{attribute 'GeneratedUsingTerminal: EL7411-0000-0016'}
{attribute addProperty BoxType "EL7411-0000-0016"}
{attribute addProperty Id "AdsAddrAT %I*AMSADDR8DcOutputShiftAT %I*DINT4DcInputShiftAT %I*DINT4Chn0AT %I*USINT1Chn1AT %I*USINT1StateAT %I*UINT2"}
{attribute addProperty CRC "1636160636"}
{attribute addProperty Size "20"}
TYPE InfoData_6185D47C :
STRUCT
	{attribute addProperty Name "AdsAddr"}
	AdsAddr AT %I* : AMSADDR;
	{attribute addProperty Name "DcOutputShift"}
	DcOutputShift AT %I* : DINT;
	{attribute addProperty Name "DcInputShift"}
	DcInputShift AT %I* : DINT;
	{attribute addProperty Name "Chn0"}
	Chn0 AT %I* : USINT;
	{attribute addProperty Name "Chn1"}
	Chn1 AT %I* : USINT;
	{attribute addProperty Name "State"}
	State AT %I* : UINT;
END_STRUCT
END_TYPE

(* stored: Version 1.2.0.0, ProductVersion 3.1.4024.9
   DUT InfoData_6185D47C: Id {43734dd9-c9c9-4af9-b1c2-67897843a21f} *)
